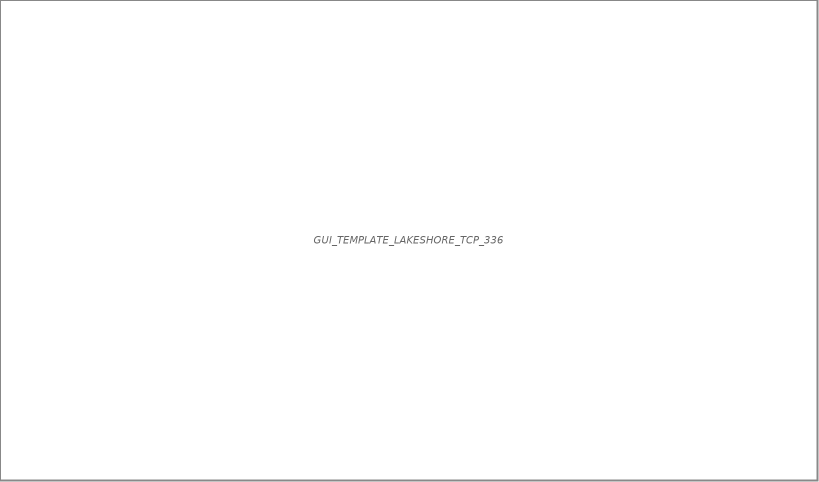
VISUALIZATION GUI_LAKESHORE_TCP_336_SIM  // 819x482
    Frame (0,0 817x480)
        shows GUI_TEMPLATE_LAKESHORE_TCP_336(m_Instance := MAIN.LS336_TCP_SIM)
END_VISUALIZATION

(* stored: Version 1.1.0.1, ProductVersion 3.1.4022.16
   Visu GUI_LAKESHORE_TCP_336_SIM: Id {36bae729-7fce-4f86-beb8-a6d4555b110c} *)
